TYPE PidParameters :
STRUCT
    Kp : LREAL;
    Ki : LREAL;
    Kd : LREAL;
END_STRUCT
END_TYPE

(* stored: Version 1.1.0.1, ProductVersion 3.1.4024.11
   DUT PidParameters: Id {68f63382-ad32-4356-9258-d4b0b1d2a26d} *)
